PROGRAM DatabaseStateMachine
VAR_INPUT
	
	bStepStart: BOOL:=TRUE;

END_VAR
	
VAR_OUTPUT
	allOutputsSet:BOOL;
END_VAR

VAR
	iState: INT;
	nextLine:ST_ProgramStruct;
	previousLine:ST_ProgramStruct;
	fbTON: TON := (PT := TIME#10S0MS);
	fbScaleValue: scaleValue;
	TempModeSwitchTrigger: F_TRIG;
		
	errorText: WSTRING(255);
	bError: BOOL;
	bSuccess: BOOL;
	iLines: UDINT;
	
	
	CalculateTemp: fbCalculateSetpoint;
	CalculateLight1: fbCalculateSetpoint;
	CalculateLight2: fbCalculateSetpoint;
	CalculateHumidity: fbCalculateSetpoint;
	
	
	
	nextLineTemp: ST_ProgramStruct;
	previousLineTemp: ST_ProgramStruct;
	
	nextLineLight1: ST_ProgramStruct;
	previousLineLight1: ST_ProgramStruct;
	
	nextLineLight2: ST_ProgramStruct;
	previousLineLight2: ST_ProgramStruct;
	
	nextLineHumidity: ST_ProgramStruct;
	previousLineHumidity: ST_ProgramStruct;
	
END_VAR

//In the case that the user switches from step mode to ramp mode, we need to set the current setpoint to the current value
//Really only needed for analog values controlled by a PID
//Like temperature, humidity...maybe CO2?

TempModeSwitchTrigger(CLK:=GVL.TempStepmode);

IF TempModeSwitchTrigger.Q THEN
	GVL.TempSetpoint:=GVL.Temp;
END_IF



CASE iState OF
	
	//Check connection
	0:
		
		fbTON(PT := TIME#1S0MS);
		allOutputsSet:=FALSE;
		IF fbTON.Q=TRUE THEN
			DBConnector();
			IF DBConnector.fbSQLDatabase.bConnected THEN
				iState:=iState+1;
				fbTON.IN:=FALSE;
			END_IF
		ELSE
			fbTON.IN:=TRUE;
		END_IF
		
		
	
	1:
		//GET TEMPERATURE
		QueryProgram(sColumn:='[Temperature]');
		IF QueryProgram.bSuccess THEN
			iState:=iState+1;
			nextLineTemp:=QueryProgram.arrRecords;
			previousLineTemp:=QueryProgram.previousLine;
			
			IF QueryProgram.bEndOfProgram THEN
				nextLineTemp.iTime:=nextLineTemp.iTime+1440;
			END_IF
			
			IF bStepStart=TRUE THEN
				GVL.TempSetpoint:=GVL.Temp;
			END_IF
			
		END_IF
		
		

	
		
	2:
		//GET LIGHT 1 LEVEL
		QueryProgram(sColumn:='[Light1]');
		
		IF QueryProgram.bSuccess THEN
				iState:=iState+1;
				nextLineLight1:=QueryProgram.arrRecords;
				previousLineLight1:=QueryProgram.previousLine;
				
				IF QueryProgram.bEndOfProgram THEN
					nextLineLight1.iTime:=nextLineLight1.iTime+1440;
				END_IF
				
		END_IF
	3:
		//GET LIGHT 2 LEVEL
		QueryProgram(sColumn:='[Light2]');
		
		IF QueryProgram.bSuccess THEN
				iState:=iState+1;
				nextLineLight2:=QueryProgram.arrRecords;
				previousLineLight2:=QueryProgram.previousLine;
				
				IF QueryProgram.bEndOfProgram THEN
					nextLineLight2.iTime:=nextLineLight2.iTime+1440;
				END_IF
				
		END_IF
	4:
		//GET HUMIDITY
		QueryProgram(sColumn:='[Humidity]');
		
		IF QueryProgram.bSuccess THEN
				iState:=iState+1;
				nextLineHumidity:=QueryProgram.arrRecords;
				previousLineHumidity:=QueryProgram.previousLine;
				
				IF QueryProgram.bEndOfProgram THEN
					nextLineHumidity.iTime:=nextLineHumidity.iTime+1440;
				END_IF
				
		END_IF
	5:
	//Success!
	allOutputsSet:=TRUE;
	iState:=0;
		

END_CASE


//Using the setpoints we just got above,
//Calculate what the target setpoint is based on
//If we're in ramp mode, step mode, what time it is, etc
CalculateTemp(
	currentValue:=GVL.Temp,
	nextSetpointValue:= nextLineTemp.Temperature, 
	nextSetpointTime:= nextLineTemp.iTime, 
	currentSetpoint:= GVL.TempSetpoint,
	previousSetpoint:=previousLineTemp.Temperature,
	previousSetpointTime:=previousLineTemp.iTime,
	stepMode:= GVL.TempStepmode, 
	setpoint=> GVL.TempSetpoint,
	bStepStart:=FALSE,
	);
	
	
CalculateLight1(
		currentValue:=GVL.Light1Percent,
		nextSetpointValue:= nextLineLight1.Light1, 
		nextSetpointTime:= nextLineLight1.iTime, 
		currentSetpoint:= GVL.Light1Percent,
		previousSetpoint:=previousLineLight1.Light1,
		previousSetpointTime:=previousLineLight1.iTime, 
		stepMode:= GVL.Light1Stepmode, 
		setpoint=> GVL.Light1Percent,
		bStepStart:=bStepStart);
		
fbScaleValue(rInputPercent:=GVL.Light1Percent,rMaxValue:=GVL.Light1Max,iScaled=>GVL.Light1Level);

CalculateLight2(
		currentValue:=GVL.Light2Percent,
		nextSetpointValue:= nextLineLight2.Light2, 
		nextSetpointTime:= nextLineLight2.iTime, 
		currentSetpoint:= GVL.Light2Percent,
		previousSetpoint:=previousLineLight2.Light2,
		previousSetpointTime:=previousLineLight2.iTime, 
		stepMode:= GVL.Light2Stepmode, 
		setpoint=> GVL.Light2Percent,
		bStepStart:=bStepStart);
		
fbScaleValue(rInputPercent:=GVL.Light2Percent,rMaxValue:=GVL.Light2Max,iScaled=>GVL.Light2Level);

CalculateHumidity(
		currentValue:=GVL.Humidity,
		nextSetpointValue:= nextLineHumidity.humidity, 
		nextSetpointTime:= nextLineHumidity.iTime, 
		currentSetpoint:= GVL.HumiditySetpoint,
		previousSetpoint:=previousLineHumidity.humidity,
		previousSetpointTime:=previousLineHumidity.iTime, 
		stepMode:= GVL.HumidityStepmode, 
		setpoint=> GVL.HumiditySetpoint,
		bStepStart:=FALSE);

END_PROGRAM

(* stored: Version 1.1.0.1, ProductVersion 3.1.4022.17
   POU DatabaseStateMachine: Id {770f277b-6e28-4759-91b2-1c985738d310}, SpecialFunc None *)
